FUNCTION_BLOCK FB_Real
VAR_INPUT
    rInput : REAL;
END_VAR
VAR_OUTPUT
    rResult : REAL;
END_VAR

rResult := rInput * 2.0;

END_FUNCTION_BLOCK

(* stored: Version 1.1.0.1, ProductVersion 3.1.4024.10
   POU FB_Real: KindOfPOU Element *)
